{attribute addProperty BoxType "EL3681-0000-0018"}
{attribute addProperty Id "StatusAT %I*Status_FB4DE8191621ValueAT %I*DINT32417"}
{attribute addProperty CRC "1634150490"}
{attribute addProperty SizeInBites "48"}
{attribute addProperty SizeInBytes "6"}
TYPE SAI_Inputs_6167285A :
STRUCT
	{attribute addProperty Name "Status"}
	Status AT %I* : Status_FB4DE819;
	{attribute addProperty Name "Value"}
	Value AT %I* : DINT;
END_STRUCT
END_TYPE

(* stored: Version 1.2.0.0, ProductVersion 3.1.4024.9
   DUT SAI_Inputs_6167285A: Id {43872e69-6aed-477b-b544-dc215ce52e5a} *)
